INTERFACE ITF_Control2_HMI_Connector_Command EXTENDS ITF_BaseControlElement_HMI_Connector_Command

END_INTERFACE

(* stored: Version 1.1.0.1
   Itf ITF_Control2_HMI_Connector_Command: Id {39e22b66-9c5b-060c-0689-a24bfcefecc3} *)
